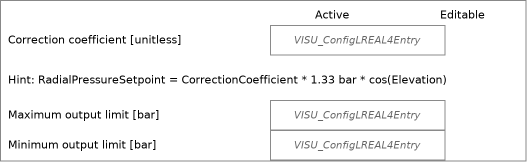
VISUALIZATION VISU_M1Config_Radial_General  // 527x162
VAR_IN_OUT
    editable : M1RadialSupportConfig;
	active : M1RadialSupportConfig;
END_VAR
    Label (270,5 125x20), "Active"
    Label (400,5 125x20), "Editable"
    Label (5,25 260x30), "Correction coefficient [unitless]"
    Frame (270,25 175x30)
        shows VISU_ConfigLREAL4Entry(active := active.correctionCoefficient, editable := editable.correctionCoefficient)
    Label (5,65 495x30), "Hint: RadialPressureSetpoint = CorrectionCoefficient * 1.33 bar * cos(Elevation)"
    Label (5,100 260x30), "Maximum output limit [bar]"
    Frame (270,100 175x30)
        shows VISU_ConfigLREAL4Entry(active := active.controllerLimitMax, editable := editable.controllerLimitMax)
    Frame (270,130 175x30)
        shows VISU_ConfigLREAL4Entry(active := active.controllerLimitMin, editable := editable.controllerLimitMin)
    Label (5,130 260x30), "Minimum output limit [bar]"
END_VISUALIZATION

(* stored: Version 1.1.0.1, ProductVersion 3.1.4019.2
   Visu VISU_M1Config_Radial_General: Id {e731a8c6-926f-49aa-a00a-5230c4cbefe6} *)
